Staubli VAL3: pow.pgx

public program pow(num x_nNumber, num x_nValue, num& x_nResult[])
  local num l_nI
begin
  //-----------------------------------------------------------------------
  //Header begin
  //Description of program
  //  This program receives 2 numbers, 1 decimal value and 1 exponent value
  //  ex: 5^2 = 25
  //  This function is similate to the Val3 function << num power(<num nX>,<num nY>) >>
  //  returns the result of nX^nY.
  //
  //Input parameters
  //  string x_nNumber :
  //    role : Decimal value
  //  string x_nValue :
  //    role : Exponent value
  //
  //Output parameters
  //  num x_nResult :
  //    role : Result of this function
  //
  //Example
  //  pow(34,5,nResult)
  //
  //History
  //  Creation : 16-04-09 - t.Gra
  //Header end
  //-----------------------------------------------------------------------
  //test 0^x = 0
  if (x_nNumber==0)
    x_nResult=0
  endIf
  //test X^0 = 1
  if round(x_nValue)==0
    x_nResult=1
    //test X^1 = X
  elseIf round(x_nValue)==1
    x_nResult=x_nNumber
  elseIf round(x_nValue)>1
    x_nResult=x_nNumber
    //calcul result loop
    for l_nI=1 to x_nValue-1
      x_nResult=x_nResult*x_nNumber
    endFor
  endIf
end
